(* IEC 61131-3 sources: ot-sentinel-lite/artifacts/icspector/baseline, 1 file *)

(* ---- conveyor_logic.st ---- *)
VAR
  Jam_Timeout : TIME := T#5s;
END_VAR
